// TIA Portal V20 export
ORGANIZATION_BLOCK "Startup"   // OB1070, LAD, Startup
TITLE = "Complete Restart"
AUTHOR : ERsystem_FA2_DH. Kim
// stored: AutoNumber false, IsIECCheckEnabled true, Namespace Unit1.Em7, SetENOAutomatically false
   VAR_INPUT
      LostRetentive : Bool;   // True if retentive data are lost
      LostRTC : Bool;   // True if date and time are lost
   END_VAR
BEGIN

REGION Network 1 (SCL): Build the Absolut Reference Designator
   // Set the Absoult Reference Designator in the Config DB
   IF LEN(IN := "Unit1.Em7.Config".em.referenceDesignator.parent) <> 0 THEN
     "Unit1.Em7.Config".em.referenceDesignator.combined := CONCAT_WSTRING(IN1 := "Unit1.Em7.Config".em.referenceDesignator.parent, IN2 := WSTRING#'.', IN3 := "Unit1.Em7.Config".em.referenceDesignator.relative);
   ELSE
     "Unit1.Em7.Config".em.referenceDesignator.combined := "Unit1.Em7.Config".em.referenceDesignator.relative;
   END_IF;
END_REGION

REGION Network 2 (SCL): Assign axes data
   //Assign axes
   "Unit1.Em7.Config".axis[1] := "BA030AZSCDR34_SepaClampnCutterAxisX";
   "Unit1.Em7.Config".axis[2] := "BA030AZSCDR35_SepaClampnCutterAxisZ";
   "Unit1.Em7.Config".axis[3] := "BA030AZSCDR36_SepaGripperAxisX";
   "Unit1.Em7.Config".axis[4] := "BA030AZSCDR37_SepaGripperAxisZ";
   "Unit1.Em7.Config".axis[5] := "BA030AZSCDR38_SepaGripperAxisC";
   "Unit1.Em7.Config".axis[6] := "BA030AZSCDR39_JRWinderRearAxisY";
   "Unit1.Em7.Config".axis[7] := "BA030AZSCDR40_JRWinderFrontAxisY";
   "Unit1.Em7.Config".axis[8] := "BA030AZSCDR41_JRWinderAxisB";
   "Unit1.Em7.Config".axis[9] := "BA030AZSDR4_JRPusherAxisZ";

   "Unit1.Em7.Config".cam[1] := "BA030AZSCDR34_SepaClampnCutterAxisXCamMain";
   "Unit1.Em7.Config".cam[2] := "BA030AZSCDR34_SepaClampnCutterAxisXCamSub";
   "Unit1.Em7.Config".cam[3] := "BA030AZSCDR35_SepaClampnCutterAxisZCamMain";
   "Unit1.Em7.Config".cam[4] := "BA030AZSCDR35_SepaClampnCutterAxisZCamSub";
   "Unit1.Em7.Config".cam[5] := "BA030AZSDR4_JRPusherAxisZMain";
   "Unit1.Em7.Config".cam[6] := "BA030AZSDR4_JRPusherAxisZSub";

   // Assign configuration data of axis

   // FB Enable
   "Unit1.Em7.HmiInterface".cmSepaClampnCutterAxisX.commands.enableMasterControl := TRUE;
   "Unit1.Em7.HmiInterface".cmSepaClampnCutterAxisZ.commands.enableMasterControl := TRUE;
   "Unit1.Em7.HmiInterface".cmSepaGripperAxisX.commands.enableMasterControl := TRUE;
   "Unit1.Em7.HmiInterface".cmSepaGripperAxisZ.commands.enableMasterControl := TRUE;
   "Unit1.Em7.HmiInterface".cmSepaGripperAxisC.commands.enableMasterControl := TRUE;
   "Unit1.Em7.HmiInterface".cmJRWinderRearAxisY.commands.enableMasterControl := TRUE;
   "Unit1.Em7.HmiInterface".cmJRWinderFrontAxisY.commands.enableMasterControl := TRUE;
   "Unit1.Em7.HmiInterface".cmJRWinderAxisB.commands.enableMasterControl := TRUE;
   "Unit1.Em7.HmiInterface".cmJRPusherAxisZ.commands.enableMasterControl := TRUE;

   // Axis 1 BA040AZSCDR34_SepaClampnCutterAxisX
   "Unit1.Em7.HmiInterface".cmSepaClampnCutterAxisX.commandConfiguration.jog.velocity := 10.0;
   "Unit1.Em7.HmiInterface".cmSepaClampnCutterAxisX.commandConfiguration.jog.acceleration := 100.0;
   "Unit1.Em7.HmiInterface".cmSepaClampnCutterAxisX.commandConfiguration.jog.deceleration := 100.0;
   "Unit1.Em7.HmiInterface".cmSepaClampnCutterAxisX.commandConfiguration.moveVelocity.velocity := 10.0;
   "Unit1.Em7.HmiInterface".cmSepaClampnCutterAxisX.commandConfiguration.moveVelocity.acceleration := 100.0;
   "Unit1.Em7.HmiInterface".cmSepaClampnCutterAxisX.commandConfiguration.moveVelocity.deceleration := 100.0;
   "Unit1.Em7.HmiInterface".cmSepaClampnCutterAxisX.commandConfiguration.posRelative.velocity := 10.0;
   "Unit1.Em7.HmiInterface".cmSepaClampnCutterAxisX.commandConfiguration.posRelative.acceleration := 100.0;
   "Unit1.Em7.HmiInterface".cmSepaClampnCutterAxisX.commandConfiguration.posRelative.deceleration := 100.0;
   "Unit1.Em7.HmiInterface".cmSepaClampnCutterAxisX.configuration.setPositions[0].name := 'waitPos';
   "Unit1.Em7.HmiInterface".cmSepaClampnCutterAxisX.configuration.setPositions[1].name := 'sepaClampnCutPos';
   "Unit1.Em7.HmiInterface".cmSepaClampnCutterAxisX.configuration.setPositions[2].name := 'winderReadyPos';
   "Unit1.Em7.HmiInterface".cmSepaClampnCutterAxisX.configuration.setPositions[3].name := 'angle90';
   "Unit1.Em7.HmiInterface".cmSepaClampnCutterAxisX.configuration.setPositions[4].name := 'angle180';
   "Unit1.Em7.HmiInterface".cmSepaClampnCutterAxisX.configuration.setPositions[5].name := 'angle270';
   "Unit1.Em7.HmiInterface".cmSepaClampnCutterAxisX.configuration.setPositions[6].name := 'angle360';
   "Unit1.Em7.HmiInterface".cmSepaClampnCutterAxisX.configuration.setPositions[7].name := 'windingDonePos';


   // Axis 2 BA040AZSCDR35_SepaClampnCutterAxisZ
   "Unit1.Em7.HmiInterface".cmSepaClampnCutterAxisZ.commandConfiguration.jog.velocity := 10.0;
   "Unit1.Em7.HmiInterface".cmSepaClampnCutterAxisZ.commandConfiguration.jog.acceleration := 100.0;
   "Unit1.Em7.HmiInterface".cmSepaClampnCutterAxisZ.commandConfiguration.jog.deceleration := 100.0;
   "Unit1.Em7.HmiInterface".cmSepaClampnCutterAxisZ.commandConfiguration.moveVelocity.velocity := 10.0;
   "Unit1.Em7.HmiInterface".cmSepaClampnCutterAxisZ.commandConfiguration.moveVelocity.acceleration := 100.0;
   "Unit1.Em7.HmiInterface".cmSepaClampnCutterAxisZ.commandConfiguration.moveVelocity.deceleration := 100.0;
   "Unit1.Em7.HmiInterface".cmSepaClampnCutterAxisZ.commandConfiguration.posRelative.velocity := 10.0;
   "Unit1.Em7.HmiInterface".cmSepaClampnCutterAxisZ.commandConfiguration.posRelative.acceleration := 100.0;
   "Unit1.Em7.HmiInterface".cmSepaClampnCutterAxisZ.commandConfiguration.posRelative.deceleration := 100.0;
   "Unit1.Em7.HmiInterface".cmSepaClampnCutterAxisZ.configuration.setPositions[0].name := 'waitPos';
   "Unit1.Em7.HmiInterface".cmSepaClampnCutterAxisZ.configuration.setPositions[1].name := 'sepaCutnClampPos';
   "Unit1.Em7.HmiInterface".cmSepaClampnCutterAxisZ.configuration.setPositions[2].name := 'winderReadyPos';
   "Unit1.Em7.HmiInterface".cmSepaClampnCutterAxisZ.configuration.setPositions[3].name := 'verticalPos';
   "Unit1.Em7.HmiInterface".cmSepaClampnCutterAxisZ.configuration.setPositions[4].name := 'horizonPos';

   // Axis 3 BA040AZSCDR36_SepaGripperAxisX
   "Unit1.Em7.HmiInterface".cmSepaGripperAxisX.commandConfiguration.jog.velocity := 10.0;
   "Unit1.Em7.HmiInterface".cmSepaGripperAxisX.commandConfiguration.jog.acceleration := 100.0;
   "Unit1.Em7.HmiInterface".cmSepaGripperAxisX.commandConfiguration.jog.deceleration := 100.0;
   "Unit1.Em7.HmiInterface".cmSepaGripperAxisX.commandConfiguration.moveVelocity.velocity := 10.0;
   "Unit1.Em7.HmiInterface".cmSepaGripperAxisX.commandConfiguration.moveVelocity.acceleration := 100.0;
   "Unit1.Em7.HmiInterface".cmSepaGripperAxisX.commandConfiguration.moveVelocity.deceleration := 100.0;
   "Unit1.Em7.HmiInterface".cmSepaGripperAxisX.commandConfiguration.posRelative.velocity := 10.0;
   "Unit1.Em7.HmiInterface".cmSepaGripperAxisX.commandConfiguration.posRelative.acceleration := 100.0;
   "Unit1.Em7.HmiInterface".cmSepaGripperAxisX.commandConfiguration.posRelative.deceleration := 100.0;
   "Unit1.Em7.HmiInterface".cmSepaGripperAxisX.configuration.setPositions[0].name := 'waitPos';
   "Unit1.Em7.HmiInterface".cmSepaGripperAxisX.configuration.setPositions[1].name := 'pickUpPOs';
   "Unit1.Em7.HmiInterface".cmSepaGripperAxisX.configuration.setPositions[2].name := 'sepaTailPos';
   "Unit1.Em7.HmiInterface".cmSepaGripperAxisX.configuration.setPositions[3].name := 'jrWinderPos';
   "Unit1.Em7.HmiInterface".cmSepaGripperAxisX.configuration.setPositions[4].name := 'turn_ngDischargePos';
   "Unit1.Em7.HmiInterface".cmSepaGripperAxisX.configuration.setPositions[5].name := 'avoidPos';
   "Unit1.Em7.HmiInterface".cmSepaGripperAxisX.configuration.setPositions[6].name := 'okDisChargePos';
   "Unit1.Em7.HmiInterface".cmSepaGripperAxisX.configuration.setPositions[7].name := 'ngSepaTailPos';
   "Unit1.Em7.HmiInterface".cmSepaGripperAxisX.configuration.setPositions[8].name := 'jrWinderZonePos';
   "Unit1.Em7.HmiInterface".cmSepaGripperAxisX.configuration.setPositions[9].name := 'gripperAxisCCollisionZonePos';
   "Unit1.Em7.HmiInterface".cmSepaGripperAxisX.configuration.setPositions[10].name := 'anodePnPZonePos';
   "Unit1.Em7.HmiInterface".cmSepaGripperAxisX.configuration.setPositions[11].name := 'pickUpBeforePos';

   // Axis 4 BA040AZSCDR37_SepaGripperAxisZ
   "Unit1.Em7.HmiInterface".cmSepaGripperAxisZ.commandConfiguration.jog.velocity := 10.0;
   "Unit1.Em7.HmiInterface".cmSepaGripperAxisZ.commandConfiguration.jog.acceleration := 100.0;
   "Unit1.Em7.HmiInterface".cmSepaGripperAxisZ.commandConfiguration.jog.deceleration := 100.0;
   "Unit1.Em7.HmiInterface".cmSepaGripperAxisZ.commandConfiguration.moveVelocity.velocity := 10.0;
   "Unit1.Em7.HmiInterface".cmSepaGripperAxisZ.commandConfiguration.moveVelocity.acceleration := 100.0;
   "Unit1.Em7.HmiInterface".cmSepaGripperAxisZ.commandConfiguration.moveVelocity.deceleration := 100.0;
   "Unit1.Em7.HmiInterface".cmSepaGripperAxisZ.commandConfiguration.posRelative.velocity := 10.0;
   "Unit1.Em7.HmiInterface".cmSepaGripperAxisZ.commandConfiguration.posRelative.acceleration := 100.0;
   "Unit1.Em7.HmiInterface".cmSepaGripperAxisZ.commandConfiguration.posRelative.deceleration := 100.0;
   "Unit1.Em7.HmiInterface".cmSepaGripperAxisZ.configuration.setPositions[0].name := 'waitPos';
   "Unit1.Em7.HmiInterface".cmSepaGripperAxisZ.configuration.setPositions[1].name := 'jrWinderPos';
   "Unit1.Em7.HmiInterface".cmSepaGripperAxisZ.configuration.setPositions[2].name := 'turnPos';
   "Unit1.Em7.HmiInterface".cmSepaGripperAxisZ.configuration.setPositions[3].name := 'jrWinderRePickUpPos';
   "Unit1.Em7.HmiInterface".cmSepaGripperAxisZ.configuration.setPositions[4].name := 'okDisChargePos';
   "Unit1.Em7.HmiInterface".cmSepaGripperAxisZ.configuration.setPositions[5].name := 'ngDischargePos';
   "Unit1.Em7.HmiInterface".cmSepaGripperAxisZ.configuration.setPositions[6].name := 'pickUpPos';

   // Axis 5 BA040AZSCDR38_SepaGripperAxisC
   "Unit1.Em7.HmiInterface".cmSepaGripperAxisC.commandConfiguration.jog.velocity := 10.0;
   "Unit1.Em7.HmiInterface".cmSepaGripperAxisC.commandConfiguration.jog.acceleration := 100.0;
   "Unit1.Em7.HmiInterface".cmSepaGripperAxisC.commandConfiguration.jog.deceleration := 100.0;
   "Unit1.Em7.HmiInterface".cmSepaGripperAxisC.commandConfiguration.moveVelocity.velocity := 10.0;
   "Unit1.Em7.HmiInterface".cmSepaGripperAxisC.commandConfiguration.moveVelocity.acceleration := 100.0;
   "Unit1.Em7.HmiInterface".cmSepaGripperAxisC.commandConfiguration.moveVelocity.deceleration := 100.0;
   "Unit1.Em7.HmiInterface".cmSepaGripperAxisC.commandConfiguration.posRelative.velocity := 10.0;
   "Unit1.Em7.HmiInterface".cmSepaGripperAxisC.commandConfiguration.posRelative.acceleration := 100.0;
   "Unit1.Em7.HmiInterface".cmSepaGripperAxisC.commandConfiguration.posRelative.deceleration := 100.0;
   "Unit1.Em7.HmiInterface".cmSepaGripperAxisC.configuration.setPositions[0].name := 'okDischargePos';
   "Unit1.Em7.HmiInterface".cmSepaGripperAxisC.configuration.setPositions[1].name := 'ngDischargePos';

   // Axis 6 BA040AZSCDR39_JRWinderRearAxisY
   "Unit1.Em7.HmiInterface".cmJRWinderFrontAxisY.commandConfiguration.jog.velocity := 10.0;
   "Unit1.Em7.HmiInterface".cmJRWinderFrontAxisY.commandConfiguration.jog.acceleration := 100.0;
   "Unit1.Em7.HmiInterface".cmJRWinderFrontAxisY.commandConfiguration.jog.deceleration := 100.0;
   "Unit1.Em7.HmiInterface".cmJRWinderFrontAxisY.commandConfiguration.moveVelocity.velocity := 10.0;
   "Unit1.Em7.HmiInterface".cmJRWinderFrontAxisY.commandConfiguration.moveVelocity.acceleration := 100.0;
   "Unit1.Em7.HmiInterface".cmJRWinderFrontAxisY.commandConfiguration.moveVelocity.deceleration := 100.0;
   "Unit1.Em7.HmiInterface".cmJRWinderFrontAxisY.commandConfiguration.posRelative.velocity := 10.0;
   "Unit1.Em7.HmiInterface".cmJRWinderFrontAxisY.commandConfiguration.posRelative.acceleration := 100.0;
   "Unit1.Em7.HmiInterface".cmJRWinderFrontAxisY.commandConfiguration.posRelative.deceleration := 100.0;
   "Unit1.Em7.HmiInterface".cmJRWinderFrontAxisY.configuration.setPositions[0].name := 'waitPos';
   "Unit1.Em7.HmiInterface".cmJRWinderFrontAxisY.configuration.setPositions[1].name := 'clampPos';

   // Axis 7 BA040AZSCDR40_JRWinderFrontAxisY
   "Unit1.Em7.HmiInterface".cmJRWinderRearAxisY.commandConfiguration.jog.velocity := 10.0;
   "Unit1.Em7.HmiInterface".cmJRWinderRearAxisY.commandConfiguration.jog.acceleration := 100.0;
   "Unit1.Em7.HmiInterface".cmJRWinderRearAxisY.commandConfiguration.jog.deceleration := 100.0;
   "Unit1.Em7.HmiInterface".cmJRWinderRearAxisY.commandConfiguration.moveVelocity.velocity := 10.0;
   "Unit1.Em7.HmiInterface".cmJRWinderRearAxisY.commandConfiguration.moveVelocity.acceleration := 100.0;
   "Unit1.Em7.HmiInterface".cmJRWinderRearAxisY.commandConfiguration.moveVelocity.deceleration := 100.0;
   "Unit1.Em7.HmiInterface".cmJRWinderRearAxisY.commandConfiguration.posRelative.velocity := 10.0;
   "Unit1.Em7.HmiInterface".cmJRWinderRearAxisY.commandConfiguration.posRelative.acceleration := 100.0;
   "Unit1.Em7.HmiInterface".cmJRWinderRearAxisY.commandConfiguration.posRelative.deceleration := 100.0;
   "Unit1.Em7.HmiInterface".cmJRWinderRearAxisY.configuration.setPositions[0].name := 'waitPos';
   "Unit1.Em7.HmiInterface".cmJRWinderRearAxisY.configuration.setPositions[1].name := 'clampPos';

   // Axis 8 BA040AZSCDR41_JRWinderAxisB
   "Unit1.Em7.HmiInterface".cmJRWinderAxisB.commandConfiguration.jog.velocity := 10.0;
   "Unit1.Em7.HmiInterface".cmJRWinderAxisB.commandConfiguration.jog.acceleration := 100.0;
   "Unit1.Em7.HmiInterface".cmJRWinderAxisB.commandConfiguration.jog.deceleration := 100.0;
   "Unit1.Em7.HmiInterface".cmJRWinderAxisB.commandConfiguration.moveVelocity.velocity := 10.0;
   "Unit1.Em7.HmiInterface".cmJRWinderAxisB.commandConfiguration.moveVelocity.acceleration := 100.0;
   "Unit1.Em7.HmiInterface".cmJRWinderAxisB.commandConfiguration.moveVelocity.deceleration := 100.0;
   "Unit1.Em7.HmiInterface".cmJRWinderAxisB.commandConfiguration.posRelative.velocity := 10.0;
   "Unit1.Em7.HmiInterface".cmJRWinderAxisB.commandConfiguration.posRelative.acceleration := 100.0;
   "Unit1.Em7.HmiInterface".cmJRWinderAxisB.commandConfiguration.posRelative.deceleration := 100.0;
   "Unit1.Em7.HmiInterface".cmJRWinderAxisB.configuration.setPositions[0].name := 'waitPos';
   "Unit1.Em7.HmiInterface".cmJRWinderAxisB.configuration.setPositions[1].name := 'angle90';
   "Unit1.Em7.HmiInterface".cmJRWinderAxisB.configuration.setPositions[2].name := 'angle180';
   "Unit1.Em7.HmiInterface".cmJRWinderAxisB.configuration.setPositions[3].name := 'angle270';
   "Unit1.Em7.HmiInterface".cmJRWinderAxisB.configuration.setPositions[4].name := 'angle360';
   "Unit1.Em7.HmiInterface".cmJRWinderAxisB.configuration.setPositions[5].name := 'angle450';
   "Unit1.Em7.HmiInterface".cmJRWinderAxisB.configuration.setPositions[6].name := 'angle540';
   "Unit1.Em7.HmiInterface".cmJRWinderAxisB.configuration.setPositions[7].name := 'winding1stPos';
   "Unit1.Em7.HmiInterface".cmJRWinderAxisB.configuration.setPositions[8].name := 'winding2ndPos';


   // Axis 9 BA040AZSDR4_JRPusherAxisZ
   "Unit1.Em7.HmiInterface".cmJRPusherAxisZ.commandConfiguration.jog.velocity := 10.0;
   "Unit1.Em7.HmiInterface".cmJRPusherAxisZ.commandConfiguration.jog.acceleration := 100.0;
   "Unit1.Em7.HmiInterface".cmJRPusherAxisZ.commandConfiguration.jog.deceleration := 100.0;
   "Unit1.Em7.HmiInterface".cmJRPusherAxisZ.commandConfiguration.moveVelocity.velocity := 10.0;
   "Unit1.Em7.HmiInterface".cmJRPusherAxisZ.commandConfiguration.moveVelocity.acceleration := 100.0;
   "Unit1.Em7.HmiInterface".cmJRPusherAxisZ.commandConfiguration.moveVelocity.deceleration := 100.0;
   "Unit1.Em7.HmiInterface".cmJRPusherAxisZ.commandConfiguration.posRelative.velocity := 10.0;
   "Unit1.Em7.HmiInterface".cmJRPusherAxisZ.commandConfiguration.posRelative.acceleration := 100.0;
   "Unit1.Em7.HmiInterface".cmJRPusherAxisZ.commandConfiguration.posRelative.deceleration := 100.0;
   "Unit1.Em7.HmiInterface".cmJRPusherAxisZ.configuration.setPositions[0].name := 'waitPos';
   "Unit1.Em7.HmiInterface".cmJRPusherAxisZ.configuration.setPositions[1].name := 'downPos';
   "Unit1.Em7.HmiInterface".cmJRPusherAxisZ.configuration.setPositions[2].name := 'verticalPos';
   "Unit1.Em7.HmiInterface".cmJRPusherAxisZ.configuration.setPositions[3].name := 'horizonPos';
END_REGION

REGION Network 3 (SCL): Assign TwoWayActuator data

   //Assign Configuration data of TwoWayActuator

   //Assign Configuration data of TwoWayActuator

   //cmSepaCutterUpDown
   "Unit1.Em7.Config".cmSepaCutterUpDown.referenceDesignator := WSTRING#'SepaCutterUpDown';
   "Unit1.Em7.Config".cmSepaCutterUpDown.disableFeedbackHomePos := FALSE;
   "Unit1.Em7.Config".cmSepaCutterUpDown.disableFeedbackWorkPos := FALSE;
   "Unit1.Em7.HmiInterface".cmSepaCutterUpDown.configuration.referenceDesignator := WSTRING#'SepaCutterUpDown';
   "Unit1.Em7.HmiInterface".cmSepaCutterUpDown.configuration.disableFeedbackHomePos := FALSE;
   "Unit1.Em7.HmiInterface".cmSepaCutterUpDown.configuration.disableFeedbackWorkPos := FALSE;

   //cmSepaClampTopUpDown
   "Unit1.Em7.Config".cmSepaClampTopUpDown.referenceDesignator := WSTRING#'SepaClampTopUpDown';
   "Unit1.Em7.Config".cmSepaClampTopUpDown.disableFeedbackHomePos := FALSE;
   "Unit1.Em7.Config".cmSepaClampTopUpDown.disableFeedbackWorkPos := FALSE;
   "Unit1.Em7.HmiInterface".cmSepaClampTopUpDown.configuration.referenceDesignator := WSTRING#'SepaClampTopUpDown';
   "Unit1.Em7.HmiInterface".cmSepaClampTopUpDown.configuration.disableFeedbackHomePos := FALSE;
   "Unit1.Em7.HmiInterface".cmSepaClampTopUpDown.configuration.disableFeedbackWorkPos := FALSE;

   //cmSepaClampBottomUpDown
   "Unit1.Em7.Config".cmSepaClampBottomUpDown.referenceDesignator := WSTRING#'SepaClampBottomUpDown';
   "Unit1.Em7.Config".cmSepaClampBottomUpDown.disableFeedbackHomePos := FALSE;
   "Unit1.Em7.Config".cmSepaClampBottomUpDown.disableFeedbackWorkPos := FALSE;
   "Unit1.Em7.HmiInterface".cmSepaClampBottomUpDown.configuration.referenceDesignator := WSTRING#'SepaClampBottomUpDown';
   "Unit1.Em7.HmiInterface".cmSepaClampBottomUpDown.configuration.disableFeedbackHomePos := FALSE;
   "Unit1.Em7.HmiInterface".cmSepaClampBottomUpDown.configuration.disableFeedbackWorkPos := FALSE;

   //cmStackGripperOpenClose
   "Unit1.Em7.Config".cmStackGripperOpenClose.referenceDesignator := WSTRING#'StackGripperOpenClose';
   "Unit1.Em7.Config".cmStackGripperOpenClose.disableFeedbackHomePos := FALSE;
   "Unit1.Em7.Config".cmStackGripperOpenClose.disableFeedbackWorkPos := FALSE;
   "Unit1.Em7.HmiInterface".cmStackGripperOpenClose.configuration.referenceDesignator := WSTRING#'StackGripperOpenClose';
   "Unit1.Em7.HmiInterface".cmStackGripperOpenClose.configuration.disableFeedbackHomePos := FALSE;
   "Unit1.Em7.HmiInterface".cmStackGripperOpenClose.configuration.disableFeedbackWorkPos := FALSE;

   //cmStackGripperFwdBwd
   "Unit1.Em7.Config".cmStackGripperFwdBwd.referenceDesignator := WSTRING#'StackGripperFwdBwd';
   "Unit1.Em7.Config".cmStackGripperFwdBwd.disableFeedbackHomePos := FALSE;
   "Unit1.Em7.Config".cmStackGripperFwdBwd.disableFeedbackWorkPos := FALSE;
   "Unit1.Em7.HmiInterface".cmStackGripperFwdBwd.configuration.referenceDesignator := WSTRING#'StackGripperFwdBwd';
   "Unit1.Em7.HmiInterface".cmStackGripperFwdBwd.configuration.disableFeedbackHomePos := FALSE;
   "Unit1.Em7.HmiInterface".cmStackGripperFwdBwd.configuration.disableFeedbackWorkPos := FALSE;

   //cmPusherRollerFwdBwd
   "Unit1.Em7.Config".cmPusherRollerFwdBwd.referenceDesignator := WSTRING#'PusherRollerFwdBwd';
   "Unit1.Em7.Config".cmPusherRollerFwdBwd.disableFeedbackHomePos := FALSE;
   "Unit1.Em7.Config".cmPusherRollerFwdBwd.disableFeedbackWorkPos := FALSE;
   "Unit1.Em7.HmiInterface".cmPusherRollerFwdBwd.configuration.referenceDesignator := WSTRING#'PusherRollerFwdBwd';
   "Unit1.Em7.HmiInterface".cmPusherRollerFwdBwd.configuration.disableFeedbackHomePos := FALSE;
   "Unit1.Em7.HmiInterface".cmPusherRollerFwdBwd.configuration.disableFeedbackWorkPos := FALSE;

   //cmJRWinderClampTopRearUpDown
   "Unit1.Em7.Config".cmJRWinderClampTopRearUpDown.referenceDesignator := WSTRING#'JRClampTopRearUpDown.';
   "Unit1.Em7.Config".cmJRWinderClampTopRearUpDown.monitoringLeavingFeedback := T#1S;
   "Unit1.Em7.Config".cmJRWinderClampTopRearUpDown.monitoringReachingFeedback := T#1S;
   "Unit1.Em7.Config".cmJRWinderClampTopRearUpDown.disableFeedbackHomePos := TRUE;
   "Unit1.Em7.Config".cmJRWinderClampTopRearUpDown.disableFeedbackWorkPos := TRUE;
   "Unit1.Em7.HmiInterface".cmJRWinderClampTopRearUpDown.configuration.referenceDesignator := WSTRING#'JRClampTopRearUpDown.';
   "Unit1.Em7.HmiInterface".cmJRWinderClampTopRearUpDown.configuration.disableFeedbackHomePos := TRUE;
   "Unit1.Em7.HmiInterface".cmJRWinderClampTopRearUpDown.configuration.disableFeedbackWorkPos := TRUE;

   //cmJRWinderClampBtmRearUpDown
   "Unit1.Em7.Config".cmJRWinderClampBtmRearUpDown.referenceDesignator := WSTRING#'JRClampBtmRearUpDown.';
   "Unit1.Em7.Config".cmJRWinderClampBtmRearUpDown.monitoringLeavingFeedback := T#1S;
   "Unit1.Em7.Config".cmJRWinderClampBtmRearUpDown.monitoringReachingFeedback := T#1S;
   "Unit1.Em7.Config".cmJRWinderClampBtmRearUpDown.disableFeedbackHomePos := TRUE;
   "Unit1.Em7.Config".cmJRWinderClampBtmRearUpDown.disableFeedbackWorkPos := TRUE;
   "Unit1.Em7.HmiInterface".cmJRWinderClampBtmRearUpDown.configuration.referenceDesignator := WSTRING#'JRClampBtmRearUpDown.';
   "Unit1.Em7.HmiInterface".cmJRWinderClampBtmRearUpDown.configuration.disableFeedbackHomePos := TRUE;
   "Unit1.Em7.HmiInterface".cmJRWinderClampBtmRearUpDown.configuration.disableFeedbackWorkPos := TRUE;

   //cmJRWinderClampTopFrontUpDown
   "Unit1.Em7.Config".cmJRWinderClampTopFrontUpDown.referenceDesignator := WSTRING#'JRClampTopFrontUpDown.';
   "Unit1.Em7.Config".cmJRWinderClampTopFrontUpDown.monitoringLeavingFeedback := T#1S;
   "Unit1.Em7.Config".cmJRWinderClampTopFrontUpDown.monitoringReachingFeedback := T#1S;
   "Unit1.Em7.Config".cmJRWinderClampTopFrontUpDown.disableFeedbackHomePos := TRUE;
   "Unit1.Em7.Config".cmJRWinderClampTopFrontUpDown.disableFeedbackWorkPos := TRUE;
   "Unit1.Em7.HmiInterface".cmJRWinderClampTopFrontUpDown.configuration.referenceDesignator := WSTRING#'JRClampTopFrontUpDown.';
   "Unit1.Em7.HmiInterface".cmJRWinderClampTopFrontUpDown.configuration.disableFeedbackHomePos := TRUE;
   "Unit1.Em7.HmiInterface".cmJRWinderClampTopFrontUpDown.configuration.disableFeedbackWorkPos := TRUE;

   //cmJRWinderClampBtmFrontUpDown
   "Unit1.Em7.Config".cmJRWinderClampBtmFrontUpDown.referenceDesignator := WSTRING#'JRClampBtmFrontUpDown.';
   "Unit1.Em7.Config".cmJRWinderClampBtmFrontUpDown.monitoringLeavingFeedback := T#1S;
   "Unit1.Em7.Config".cmJRWinderClampBtmFrontUpDown.monitoringReachingFeedback := T#1S;
   "Unit1.Em7.Config".cmJRWinderClampBtmFrontUpDown.disableFeedbackHomePos := TRUE;
   "Unit1.Em7.Config".cmJRWinderClampBtmFrontUpDown.disableFeedbackWorkPos := TRUE;
   "Unit1.Em7.HmiInterface".cmJRWinderClampBtmFrontUpDown.configuration.referenceDesignator := WSTRING#'JRClampBtmFrontUpDown.';
   "Unit1.Em7.HmiInterface".cmJRWinderClampBtmFrontUpDown.configuration.disableFeedbackHomePos := TRUE;
   "Unit1.Em7.HmiInterface".cmJRWinderClampBtmFrontUpDown.configuration.disableFeedbackWorkPos := TRUE;
END_REGION
END_ORGANIZATION_BLOCK
